(* CODESYS project PWM.project
   Title: PWM
   Version: 0.0.0.0
   Author: MustafaZahid

Project tree, tasks and I/O mapping:
  MyController : TM241C24T/U, Schneider Electric, order no. TM241C24T/U, version 4.0.6.18
    application Application
      task MAST (cyclic, interval 20 ms, priority 15, watchdog 100 ms x 1) calls POU
      global variables GVL
      program POU [LD]
    DI : Digital Inputs, Schneider Electric, version 4.0.6.18
        input  iwDI_IW0 : WORD  // IW0
        input  ibDI_IB1 : BYTE  // IB1
    DQ : Digital Outputs, Schneider Electric, version 4.0.6.18
        settings: Outputs Usage = 1
        output qwDQ_QW0 : WORD  // QW0
        output qbDQ_QB1 : BYTE  // QB1
    Counters : Counters, Schneider Electric, version 4.0.6.18
    Pulse_Generators : Pulse Generators, Schneider Electric, version 4.0.6.18
        settings: Instance name = 'PWM_0'; A output History = 'old=-1 new=0'; Temporary Instance name = 'PWM_0'
    Cartridge_1 : Cartridge, Schneider Electric, version 4.0.6.18
    IO_Bus : IO bus - TM3, Schneider Electric, version 4.0.6.18
    COM_Bus : COM bus, Schneider Electric, version 4.0.6.18
    Serial_Line_1 : Serial line, Schneider Electric, version 4.0.6.18
      SoMachine_Network_Manager : SoMachine-Network Manager, Schneider Electric, version 4.0.0.2
    Serial_Line_2 : Serial line, Schneider Electric, version 4.0.6.18
      Modbus_Manager : Modbus Manager, Schneider Electric, version 4.0.0.2
*)

// MyController/Application/GVL
VAR_GLOBAL
END_VAR

// MyController/Application/POU
PROGRAM POU
VAR
	PWM_EN: BOOL;
	PWM_F_EN: BOOL;
	PWM_SYNC: BOOL;
	PWM_F_SYNC: BOOL;
	PWM_Freq: DWORD;
	PWM_Duty: UINT;
END_VAR

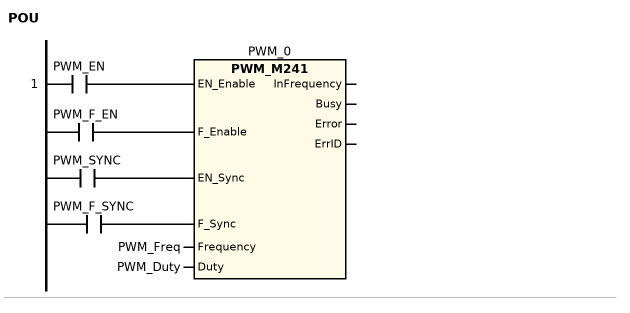
// NETWORK 1
PWM_0(
    EN_Enable := PWM_EN,
    F_Enable := PWM_F_EN,
    EN_Sync := PWM_SYNC,
    F_Sync := PWM_F_SYNC,
    Frequency := PWM_Freq,
    Duty := PWM_Duty); // PWM_M241

END_PROGRAM
